{attribute 'qualified_only'}
{attribute 'strict'}
{attribute 'to_string'}
TYPE E_SeqInit :
(
	GENERAL := 0,
	BIAS,
	CALIBRATED,
	DONE
);
END_TYPE

(* stored: Version 1.1.0.1, ProductVersion 3.1.4024.12
   DUT E_SeqInit: Id {902d633e-d1e1-4844-878f-3549c7ec2eb2} *)
